PROGRAM S_LoadWafer
VAR_INPUT
	bInit				:BOOL:=FALSE;// 初始化状态 busy/done/errDone
	bTrig				:BOOL:=FALSE;// 执行触发 信号
	bReset				:BOOL:=FALSE;// 报错 复位
	bPause				:BOOL:=FALSE;// 暂停 运行
	bStop				:BOOL:=FALSE;// 停止 运行
	bAbort				:BOOL:=FALSE;// 中止 运行
	
END_VAR
VAR_OUTPUT
	busy				:BOOL;
	done				:BOOL;
	errDone				:BOOL;
END_VAR
VAR
	actStep				:ActStepBase;
END_VAR
VAR
	i: INT;
	t1:ton;
	t2:ton;
	t3:ton;
	notchoose:BOOL;
	timeOutTime:TIME:= T#60S;
	ventTime:TIME:=T#20S;
END_VAR

busy:=actStep.isBusy();
done:=actStep.isDone();
errDone:=actStep.isError();
actStep.Act_Pause(pause:=bPause);

IF bTrig THEN
	bTrig:=FALSE;
	IF NOT busy THEN
		actStep.Act_ex();
	END_IF
END_IF

//状态复位
IF bInit THEN
	bInit:=FALSE;
	Act_init_status();
END_IF

IF bAbort OR bStop THEN
	bAbort:=FALSE;
	bStop:=FALSE;
	Act_init_status();
	actStep.toZeroStep();
	gShowLogTextTitle:='NON';
END_IF
ActionRun(tempActStep:=actStep);

(*
---Trigger action
*)
METHOD Act_Ex : BOOL
VAR_INPUT
END_VAR
IF NOT busy THEN
	actStep.Act_ex();
	Act_Ex:=TRUE;
ELSE
	Act_Ex:=FALSE;
END_IF
END_METHOD

(*
---功能: 状态复位 busy/done/errDone;
*)
METHOD Act_Init_Status
VAR_INPUT
END_VAR
actStep.Act_Init();
END_METHOD

METHOD PRIVATE ActionRun
VAR_INPUT
	tempActStep:ITFActStep;
END_VAR
VAR_STAT//此处定义静态变量, 保证每次进入该函数时能够在线监控当前值
	tempStep:DINT;
END_VAR
tempStep:=tempActStep.getStep();
CASE tempStep OF
0:
	IF tempActStep.isEx() THEN
		tempActStep.setBusyFlag();
		tempActStep.toBeginStep();
	END_IF
	t1(IN:= FALSE );
	t2(IN:= FALSE );
	t3(IN:= FALSE );
10:
	gShowLogTextTitle:='Load Wafer';
	IF gRunningState<>RunningStatus.eErrorState THEN
		tempActStep.addStep(10,FALSE);
	ELSE
		error_Trigger(105);
		IF gCtrlMode=ControlMode.eManualCtrMode THEN
			tempActStep.toErrDoneStep();
		END_IF
	END_IF
20:
	IF ControlMode.eManualCtrMode=gCtrlMode THEN
//		S_WaferCheckPOU.Act_Init_Status();
//		S_WaferCheckPOU.Act_Ex();
		tempActStep.addStep(10,FALSE);
	ELSIF( ControlMode.eAutoCtrMode=gCtrlMode) THEN
		tempActStep.addStep(10,FALSE);
	ELSE
		tempActStep.toErrDoneStep();
	END_IF
30:
	tempActStep.addStep(10,FALSE);
40:
	tempActStep.addStep(10,TRUE);
50:
	tempActStep.addStep(10,FALSE);
60:
	S_RoughPumping.Act_Init_Status();
	S_RoughPumping.Act_Ex();
	tempActStep.addStep(10,FALSE);
70:
	IF S_RoughPumping.done THEN
		gShowLogTextTitle:='Load Wafer';
		tempActStep.addStep(10,FALSE);
	END_IF
	IF S_RoughPumping.errDone THEN
		tempActStep.toStep(40,FALSE);
	END_IF
80:
	tempActStep.addStep(20,TRUE);
100:
	IF gWaferMemoryState=1 THEN// 腔体有晶圆
		gRunningLog.append(CONCAT('Load Wafer POU Run:',DINT_TO_STRING(tempStep)));
		gRunningLog.append('Load Wafer POU Run: Wafer In Chamber ');
		tempActStep.toStep(590,FALSE);
	ELSE// 腔体无晶圆
		gRunningLog.append(CONCAT('Load Wafer POU Run:',DINT_TO_STRING(tempStep)));
		gRunningLog.append('Load Wafer POU Run: Wafer OutSide Chamber ');
		IF NOT gICP.I_WaferCheck THEN
			tempActStep.addStep(10,FALSE);// 手臂上无晶圆
			gRunningLog.append('Load Wafer POU Run: There are wafers on the arm ');
		ELSE
			gRunningLog.append('Load Wafer POU Run: There are not wafers on the arm ');
			tempActStep.toStep(200,FALSE);// 手臂上有晶圆
		END_IF
	END_IF
110:
	tempActStep.addStep(5,TRUE);
115:
	IF  gICP.GateDoorValve.Act_Retract() AND 
	    gICP.SlowPummingValve.Act_Retract() AND 
	    gICP.FastPummingValve.Act_Retract() THEN
		gRunningLog.append(CONCAT('Load Wafer POU Run:',DINT_TO_STRING(tempStep)));
		gRunningLog.append('Load Wafer POU Run:LoadLock Close');
		tempActStep.addStep(5,FALSE);
	END_IF
120:
	IF gICP.GateDoorValve.Get_Done_Ret() AND gICP.GateDoorRetSensor AND
	   gICP.SlowPummingValve.Get_Done_Ret() AND NOT gICP.SlowPummingExtRelay AND
	   gICP.FastPummingValve.Get_Done_Ret() AND NOT gICP.FastPummingExtRelay THEN
	   gRunningLog.append(CONCAT('Load Wafer POU Run:',DINT_TO_STRING(tempStep)));
	   gRunningLog.append('Load Wafer POU Run:LoadLock Close Done');
		tempActStep.addStep(10,FALSE);
	END_IF
130:
	IF gICP.VentValve.Act_Extend() THEN
		gRunningLog.append(CONCAT('Load Wafer POU Run:',DINT_TO_STRING(tempStep)));
		gRunningLog.append('Load Wafer POU Run:Vent Open');
		tempActStep.addStep(10,FALSE);
	END_IF
140:
	IF gICP.VentValve.Get_Done_Ext() THEN
		gRunningLog.append(CONCAT('Load Wafer POU Run:',DINT_TO_STRING(tempStep)));
		gRunningLog.append('Load Wafer POU Run:Vent Open Done');
		tempActStep.addStep(10,FALSE);
	END_IF
150:
	t2(IN:=gICP.LoadLockGauge.outputValue>gATMPressure,PT:=ventTime);
	IF t2.Q OR NOT gICP.I_LLSwitch THEN
		gRunningLog.append(CONCAT('Load Wafer POU Run:',DINT_TO_STRING(tempStep)));
		gRunningLog.append(CONCAT('Load Wafer POU Run:LL Vent Pressure Arrive：',REAL_TO_STRING(gICP.LoadLockGauge.outputValue)));
		t1(IN:= FALSE );
		t2(IN:= FALSE );
		t3(IN:= FALSE );
		tempActStep.addStep(10,FALSE);
		RETURN;
	END_IF
	t1(IN:= TRUE,PT:=timeOutTime );
	IF t1.Q THEN
		t1(IN:= FALSE );
		t2(IN:= FALSE );
		t3(IN:= FALSE );
		error_Trigger(110);
		tempActStep.toStep(110,FALSE);
		RETURN;
	END_IF
160:
	tempActStep.addStep(10,TRUE);
170:
	IF gICP.VentValve.Act_Retract() THEN
		gRunningLog.append(CONCAT('Load Wafer POU Run:',DINT_TO_STRING(tempStep)));
		gRunningLog.append('Load Wafer POU Run:Vent Close');
		tempActStep.addStep(10,FALSE);
	END_IF
180:
	IF gICP.GateDoorValve.Get_Done_Ret() THEN
		gRunningLog.append(CONCAT('Load Wafer POU Run:',DINT_TO_STRING(tempStep)));
		gRunningLog.append('Load Wafer POU Run:Vent Close Done');
		tempActStep.addStep(10,FALSE);
	END_IF
190:
	t1(IN:=TRUE,PT:=T#1S);
	IF t1.Q THEN
		t1(IN:= FALSE );
		t2(IN:= FALSE );
		t3(IN:= FALSE );
		gRunningLog.append(CONCAT('Load Wafer POU Run:',DINT_TO_STRING(tempStep)));
		gRunningLog.append('Load Wafer POU Run:Wait for the wafer to be placed');
		tempActStep.addStep(10,FALSE);
	END_IF
200:
	t2(IN:=gICP.I_WaferCheck AND gICP.I_LLSwitch,PT:=T#5S);// 放入晶圆，且关上盖子
	IF t2.Q THEN
		gRunningLog.append('Load Wafer POU Run:Place the wafer and close the lid');
		t1(IN:= FALSE );
		t2(IN:= FALSE );
		t3(IN:= FALSE );
		tempActStep.addStep(10,FALSE);
		RETURN;
	END_IF
	t3(IN:=TRUE,PT:=timeOutTime);
	IF t3.Q THEN
		error_Trigger(110);
		t1(IN:= FALSE );
		t2(IN:= FALSE );
		t3(IN:= FALSE );
		tempActStep.tostep(160,FALSE);
	END_IF
210:
	tempActStep.addStep(5,TRUE);
215:
	t2(IN:=gICP.LoadLockGauge.outputValue<gRoughtPumVaccum,PT:=T#2S);
	IF t2.Q THEN
		gRunningLog.append(CONCAT('Load Wafer POU Run:',DINT_TO_STRING(tempStep)));
		gRunningLog.append(CONCAT('Load Wafer POU Run:LL Pumping Pressure Arrive：',REAL_TO_STRING(gICP.LoadLockGauge.outputValue)));
		t1(IN:= FALSE );
		t2(IN:= FALSE );
		t3(IN:= FALSE );
		tempActStep.tostep(310,FALSE);
		RETURN;
	END_IF
	t3(IN:=TRUE,PT:=T#3S);
	IF t3.Q THEN
		t1(IN:= FALSE );
		t2(IN:= FALSE );
		t3(IN:= FALSE );
		IF  gICP.VentValve.Act_Retract() AND 
			gICP.ForlinLineValve.Act_Retract() AND 
			gICP.RoughValve.Act_Retract() THEN
			gRunningLog.append(CONCAT('Load Wafer POU Run:',DINT_TO_STRING(tempStep)));
			gRunningLog.append('Load Wafer POU Run:LL Pumping(Close Vent\Forline\Rough Valve)');
			tempActStep.addStep(5,FALSE);
		END_IF
	END_IF
220:
	IF gICP.VentValve.Get_Done_Ret() AND NOT gICP.VentExtRelay AND
	   gICP.ForlinLineValve.Get_Done_Ret() AND NOT gICP.ForlinLineValveExtRelay AND
	   gICP.RoughValve.Get_Done_Ret() AND NOT gICP.RoughValveExtRelay THEN
	   gRunningLog.append(CONCAT('Load Wafer POU Run:',DINT_TO_STRING(tempStep)));
	   gRunningLog.append('Load Wafer POU Run:LL Pumping(Vent\Forline\Rough Valve Close Done)');
		tempActStep.addStep(10,FALSE);
	END_IF
230://////////////准备抽LoadLock
	tempActStep.addStep(10,FALSE);
240:
	tempActStep.addStep(10,TRUE);
250:
	IF gICP.SlowPummingValve.Act_Extend() AND gICP.FastPummingValve.Act_Retract() THEN
		gRunningLog.append(CONCAT('Load Wafer POU Run:',DINT_TO_STRING(tempStep)));
		gRunningLog.append('Load Wafer POU Run:LL Rough Pumping(SlowPum Valve Open \ FastPum Valve Close)');
		tempActStep.addStep(10,FALSE);
	END_IF
260:
	IF gICP.SlowPummingValve.Get_Done_Ext() AND gICP.FastPummingValve.Get_Done_Ret() THEN
		gRunningLog.append(CONCAT('Load Wafer POU Run:',DINT_TO_STRING(tempStep)));
		gRunningLog.append('Load Wafer POU Run:LL Rough Pumping(SlowPum Valve Open Done\ FastPum Valve Close Done)');
		tempActStep.addStep(10,FALSE);
	END_IF
270:
	t2(IN:=gICP.LoadLockGauge.outputValue<gLoadLockPumSVaccum,PT:=T#2S);
	IF t2.Q THEN
		gRunningLog.append(CONCAT('Load Wafer POU Run:',DINT_TO_STRING(tempStep)));
		gRunningLog.append(CONCAT('Load Wafer POU Run:LL Rough Pumping Pressure Arrive：',REAL_TO_STRING(gICP.LoadLockGauge.outputValue)));
		t1(IN:= FALSE );
		t2(IN:= FALSE );
		t3(IN:= FALSE );
		tempActStep.addStep(10,FALSE);
	END_IF
280:
	IF gICP.SlowPummingValve.Act_Retract() AND gICP.FastPummingValve.Act_Extend() THEN
		gRunningLog.append(CONCAT('Load Wafer POU Run:',DINT_TO_STRING(tempStep)));
		gRunningLog.append('Load Wafer POU Run:LL Fast Pumping(SlowPum Valve Close \ FastPum Valve Open)');
		tempActStep.addStep(10,FALSE);
	END_IF
290:
	IF gICP.SlowPummingValve.Get_Done_Ret() AND gICP.FastPummingValve.Get_Done_Ext() THEN
		gRunningLog.append(CONCAT('Load Wafer POU Run:',DINT_TO_STRING(tempStep)));
		gRunningLog.append('Load Wafer POU Run:LL Fast Pumping(SlowPum Valve Close Done\ FastPum Valve Open Done)');
		tempActStep.addStep(10,FALSE);
	END_IF
300:
	t2(IN:=gICP.LoadLockGauge.outputValue<gRoughtPumVaccum,PT:=T#2S);
	IF t2.Q THEN
		gRunningLog.append(CONCAT('Load Wafer POU Run:',DINT_TO_STRING(tempStep)));
		gRunningLog.append(CONCAT('Load Wafer POU Run:LL Fast Pumping Pressure Arrive：',REAL_TO_STRING(gICP.LoadLockGauge.outputValue)));
		t1(IN:= FALSE );
		t2(IN:= FALSE );
		t3(IN:= FALSE );
		tempActStep.addStep(10,FALSE);
	END_IF
310:
	tempActStep.addStep(10,TRUE);
320:
	IF gICP.SlowPummingValve.Act_Retract() AND gICP.FastPummingValve.Act_Retract() THEN
		gRunningLog.append(CONCAT('Load Wafer POU Run:',DINT_TO_STRING(tempStep)));
		gRunningLog.append('Load Wafer POU Run:LL Fast Pumping(SlowPum Valve Close \ FastPum Valve Close)');
		tempActStep.addStep(10,FALSE);
	END_IF
330:
	IF gICP.SlowPummingValve.Get_Done_Ret() AND gICP.FastPummingValve.Get_Done_Ret() THEN
		gRunningLog.append(CONCAT('Load Wafer POU Run:',DINT_TO_STRING(tempStep)));
		gRunningLog.append('Load Wafer POU Run:LL Fast Pumping(SlowPum Valve Close Done\ FastPum Valve Close Done)');
		tempActStep.addStep(10,FALSE);
	END_IF
340:
	tempActStep.addStep(2,TRUE);
342:
	IF gICP.PDV.Act_Retract() THEN
		gRunningLog.append(CONCAT('Load Wafer POU Run:',DINT_TO_STRING(tempStep)));
		gRunningLog.append('Load Wafer POU Run:PDV Close');
		tempActStep.addStep(2,FALSE);
	END_IF
344:
	IF gICP.PDV.Get_Done_Ret() OR gICP.PDVCloseSensor THEN
		gRunningLog.append(CONCAT('Load Wafer POU Run:',DINT_TO_STRING(tempStep)));
		gRunningLog.append('Load Wafer POU Run:PDV Close Done');
		tempActStep.addStep(2,FALSE);
	END_IF
346:
	tempActStep.addStep(4,TRUE);
350:
	IF gICP.GateDoorValve.Act_Extend() THEN
		gRunningLog.append(CONCAT('Load Wafer POU Run:',DINT_TO_STRING(tempStep)));
		gRunningLog.append('Load Wafer POU Run:Gate Door Open');
		tempActStep.addStep(10,FALSE);
	END_IF
360:
	IF gICP.GateDoorValve.Get_Done_Ext() AND gICP.GateDoorExtSensor THEN
		gRunningLog.append(CONCAT('Load Wafer POU Run:',DINT_TO_STRING(tempStep)));
		gRunningLog.append('Load Wafer POU Run:Gate Door Open Done');
		tempActStep.addStep(10,FALSE);
	END_IF
370:
	IF gICP.ElectrodeCyl.Act_Retract() AND gICP.LiftPinCyl.Act_Retract() THEN
		gRunningLog.append(CONCAT('Load Wafer POU Run:',DINT_TO_STRING(tempStep)));
		gRunningLog.append('Load Wafer POU Run:ElectrodeCyl&LiftPinCyl Down');
		tempActStep.addStep(10,FALSE);
	END_IF
380:
	IF gICP.ElectrodeCyl.Get_Done_Ret() AND gICP.LiftPinCyl.Get_Done_Ret() THEN
		gRunningLog.append(CONCAT('Load Wafer POU Run:',DINT_TO_STRING(tempStep)));
		gRunningLog.append('Load Wafer POU Run:ElectrodeCyl&LiftPinCyl Down Done');
		tempActStep.addStep(10,FALSE);
	END_IF
390:
	tempActStep.addStep(10,TRUE);
400:
	IF gICP.ARM.Act_IN_Auto() THEN
		gRunningLog.append(CONCAT('Load Wafer POU Run:',DINT_TO_STRING(tempStep)));
		gRunningLog.append('Load Wafer POU Run:ARM IN');
		tempActStep.addStep(10,FALSE);
	END_IF
410:
	IF NOT gICP.I_ARMHome THEN// 手臂当前不应该在原点位置
		gRunningLog.append(CONCAT('Load Wafer POU Run:',DINT_TO_STRING(tempStep)));
		gRunningLog.append('Load Wafer POU Run:ARM Running');
		tempActStep.addStep(10,FALSE);
	END_IF
420:
	t2(IN:=gICP.ARM.Get_Done_IN() AND NOT(gICP.ARM.busy OR gICP.ARM.jogBusy),PT:=T#3S);
	IF t2.Q  THEN
		t1(IN:= FALSE );
		t2(IN:= FALSE );
		t3(IN:= FALSE );
		gRunningLog.append(CONCAT('Load Wafer POU Run:',DINT_TO_STRING(tempStep)));
		gRunningLog.append('Load Wafer POU Run:ARM IN Done');
		tempActStep.addStep(10,FALSE);
		RETURN;
	END_IF
	t1(IN:=TRUE,PT:=T#30S);
	IF t1.Q THEN
		t1(IN:= FALSE );
		t2(IN:= FALSE );
		t3(IN:= FALSE );
		error_Trigger(111);
		tempActStep.toStep(390,FALSE);// 报错
		RETURN;
	END_IF
430:
	tempActStep.addStep(10,TRUE);
440:
	IF gICP.LiftPinCyl.Act_Extend() THEN
		tempActStep.addStep(10,FALSE);
	END_IF
450:
	IF gICP.LiftPinCyl.Get_Done_Ext() AND gICP.LiftPinExtSensor THEN
		gRunningLog.append(CONCAT('Load Wafer POU Run:',DINT_TO_STRING(tempStep)));
		gRunningLog.append('Load Wafer POU Run:LiftPinCyl UP And Remember Wafer Memory ');
		// 记忆状态更新
		gWaferMemoryState:=1;
		ups_CX51X0.Act_Wrtie();
		tempActStep.addStep(10,FALSE);
	END_IF
460:
	tempActStep.addStep(10,TRUE);
470:
	IF gICP.ARM.Act_HOME_Auto() THEN
		gRunningLog.append(CONCAT('Load Wafer POU Run:',DINT_TO_STRING(tempStep)));
		gRunningLog.append('Load Wafer POU Run:ARM Home ');
		tempActStep.addStep(10,FALSE);
	END_IF
480:
	IF gICP.ARM.Get_Done_HOME() AND gICP.I_ARMHome AND NOT(gICP.ARM.busy OR gICP.ARM.jogBusy) THEN// 手臂当前不应该在原点位置
		gRunningLog.append(CONCAT('Load Wafer POU Run:',DINT_TO_STRING(tempStep)));
		gRunningLog.append('Load Wafer POU Run:ARM Home Done');
		tempActStep.addStep(10,FALSE);
	END_IF
490:
	t2(IN:=TRUE,PT:=T#3S);
	IF t2.Q THEN
		t1(IN:= FALSE );
		t2(IN:= FALSE );
		t3(IN:= FALSE );
		tempActStep.addStep(10,FALSE);
		RETURN;
	END_IF
500:
	tempActStep.addStep(10,TRUE);
510:
	IF gICP.GateDoorValve.Act_Retract() AND gICP.LiftPinCyl.Act_Retract() THEN
		gRunningLog.append(CONCAT('Load Wafer POU Run:',DINT_TO_STRING(tempStep)));
		gRunningLog.append('Load Wafer POU Run:Gate Door Close And LiftPinCyl Down');
		tempActStep.addStep(10,FALSE);
	END_IF
520:
	IF gICP.GateDoorValve.Get_Done_Ret() AND gICP.GateDoorRetSensor AND
	   gICP.LiftPinCyl.Get_Done_Ret() AND gICP.LiftPinRetSensor THEN
	   gRunningLog.append(CONCAT('Load Wafer POU Run:',DINT_TO_STRING(tempStep)));
	   gRunningLog.append('Load Wafer POU Run:Gate Door Close Done And LiftPinCyl Down Done');
		tempActStep.addStep(10,FALSE);
	END_IF
530:
	tempActStep.addStep(10,TRUE);
540:
	IF gICP.ForlinLineValve.Act_Extend() THEN
		gRunningLog.append(CONCAT('Load Wafer POU Run:',DINT_TO_STRING(tempStep)));
		gRunningLog.append('Load Wafer POU Run:ForLine Valve Open');
		tempActStep.addStep(10,FALSE);
	END_IF
550:
	IF gICP.ForlinLineValve.Get_Done_Ext() THEN
		gRunningLog.append(CONCAT('Load Wafer POU Run:',DINT_TO_STRING(tempStep)));
		gRunningLog.append('Load Wafer POU Run:ForLine Valve Open Done');
		tempActStep.addStep(10,FALSE);
	END_IF
560:
	tempActStep.addStep(10,TRUE);
570:
	IF gICP.PDV.Act_Open() THEN
		gRunningLog.append(CONCAT('Load Wafer POU Run:',DINT_TO_STRING(tempStep)));
		gRunningLog.append('Load Wafer POU Run:PDV Open');
		tempActStep.addStep(10,FALSE);
	END_IF
580:
	IF gICP.PDV.Get_Done_Ext() OR gICP.PDVOpenSensor THEN
		gRunningLog.append(CONCAT('Load Wafer POU Run:',DINT_TO_STRING(tempStep)));
		gRunningLog.append('Load Wafer POU Run:PDV Open Done');
		tempActStep.addStep(10,FALSE);
	END_IF
590:
	// 记忆状态更新
	gWaferMemoryState:=1;
	ups_CX51X0.Act_Wrtie();
	gRunningLog.append(CONCAT('Load Wafer POU Run:',DINT_TO_STRING(tempStep)));
	gRunningLog.append('Load Wafer POU Run:----Finish----');
	tempActStep.toDoneStep();
1000:
	tempActStep.toDoneStep();

60000://Done
	tempActStep.setDoneFlag();
	tempActStep.toZeroStep();
	
65000://Error
	tempActStep.setErrDoneFlag();
	tempActStep.toZeroStep();
	IF gICP.VentExtRelay THEN
		gICP.VentValve.Act_Retract();
	END_IF
END_CASE
END_METHOD

END_PROGRAM

(* stored: Version 1.1.0.1, ProductVersion 3.1.4024.12
   POU S_LoadWafer: Id {82a0232f-04ff-4bdb-8459-9a013dba7728}, SpecialFunc None
   Folder Private: Id {a175c7e9-f3fe-49e0-beee-76dc86a58095}
   Method Act_Ex: Id {6b613451-6d6c-4cbb-be84-a4989bff788b}
   Method Act_Init_Status: Id {703970f9-4130-4985-9921-7ee8730f71f4}
   Method ActionRun: Id {17b0de09-3fb2-4c97-8a30-333a04f8ee9a} *)
